{attribute addProperty BoxType "EK1122-0000-0018"}
{attribute addProperty Id "Beckhoff_EL29xxsub_EK1100EK1100_179A0949162"}
{attribute addProperty CRC "3909730180"}
{attribute addProperty SizeInBites "16"}
{attribute addProperty SizeInBytes "2"}
TYPE Beckhoff_EL29xxEK1122_E909BF84 EXTENDS EK1122_179A0949 :
STRUCT
	{attribute addProperty Name "Beckhoff_EL29xxsub_EK1100"}
	Beckhoff_EL29xxsub_EK1100 : EK1100_179A0949;
END_STRUCT
END_TYPE

(* stored: Version 1.2.0.0, ProductVersion 3.1.4024.9
   DUT Beckhoff_EL29xxEK1122_E909BF84: Id {53b2f0a8-d117-49f1-ae48-fd696b134190} *)
